PROGRAM C07_EtherCATDiagnostic
VAR
	(*sEtherCATMasterAmsNetID	: T_AmsNetID;*)
	fbBlink							: FB_Blink;

	fbGetDeviceNetId				: IOF_GetDeviceNetId;

	fbEcGetAllSlaveStates			: FB_EcGetAllSlaveStates;
	aSlaveStates					: ARRAY[0..cMAX_ETHERCAT_SLAVES] OF ST_EcSlaveState;

	fbEcGetConfSlaves				: FB_EcGetConfSlaves;
	aEcConfSlaveInfo 				: ARRAY[0..cMAX_ETHERCAT_SLAVES] OF ST_EcSlaveConfigData;

	fbEtherCATStatus				: FB_CX_EtherCATStatus;
END_VAR

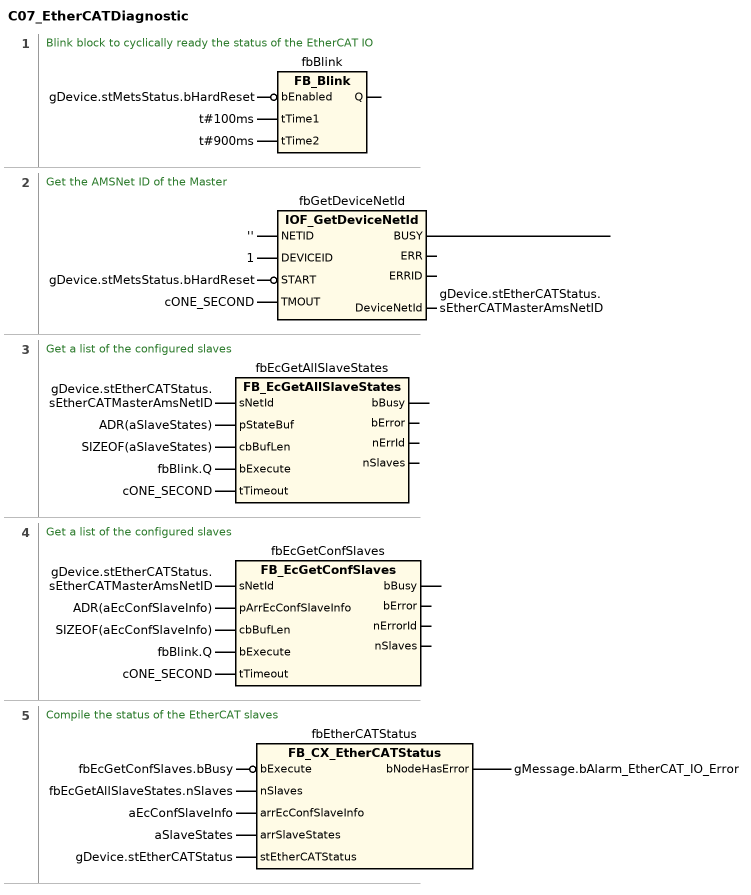
// NETWORK 1
// Blink block to cyclically ready the status of the EtherCAT IO
fbBlink(bEnabled := NOT gDevice.stMetsStatus.bHardReset, tTime1 := t#100ms, tTime2 := t#900ms); // FB_Blink

// NETWORK 2
// Get the AMSNet ID of the Master
fbGetDeviceNetId(
    NETID := '',
    DEVICEID := 1,
    START := NOT gDevice.stMetsStatus.bHardReset,
    TMOUT := cONE_SECOND,
    DeviceNetId => gDevice.stEtherCATStatus.sEtherCATMasterAmsNetID); // IOF_GetDeviceNetId

// NETWORK 3
// Get a list of the configured slaves
fbEcGetAllSlaveStates(
    sNetId := gDevice.stEtherCATStatus.sEtherCATMasterAmsNetID,
    pStateBuf := ADR(aSlaveStates),
    cbBufLen := SIZEOF(aSlaveStates),
    bExecute := fbBlink.Q,
    tTimeout := cONE_SECOND); // FB_EcGetAllSlaveStates

// NETWORK 4
// Get a list of the configured slaves
fbEcGetConfSlaves(
    sNetId := gDevice.stEtherCATStatus.sEtherCATMasterAmsNetID,
    pArrEcConfSlaveInfo := ADR(aEcConfSlaveInfo),
    cbBufLen := SIZEOF(aEcConfSlaveInfo),
    bExecute := fbBlink.Q,
    tTimeout := cONE_SECOND); // FB_EcGetConfSlaves

// NETWORK 5
// Compile the status of the EtherCAT slaves
fbEtherCATStatus(
    bExecute := NOT fbEcGetConfSlaves.bBusy,
    nSlaves := fbEcGetAllSlaveStates.nSlaves,
    arrEcConfSlaveInfo := aEcConfSlaveInfo,
    arrSlaveStates := aSlaveStates,
    stEtherCATStatus := gDevice.stEtherCATStatus); // FB_CX_EtherCATStatus
gMessage.bAlarm_EtherCAT_IO_Error := fbEtherCATStatus.bNodeHasError;

END_PROGRAM

(* stored: Version 1.1.0.1
   POU C07_EtherCATDiagnostic: Id {f4360ef3-04b8-46ac-a08a-dd1bd9c2f069}, SpecialFunc None *)
